// TwinCAT 3 PLC project Builder2
// ProgramVersion: 3.1.4023.0
// libraries:
//   Tc2_Standard, * (Beckhoff Automation GmbH)
//   Tc2_System, * (Beckhoff Automation GmbH)
//   Tc3_Module, * (Beckhoff Automation GmbH)
//   VisuSymbols,3.5.10.0,System
// project tree:
//   / Class Diagram_1.TcCD (not stored), ConcreteBuilder.TcPOU, Director.TcPOU, GlobalTextList.TcGTLO, ITF_Builder.TcIO, PlcTask.TcTTO, Product.TcPOU, Visualization Manager.TcVMO (not stored)
//   POUs/ MAIN.TcPOU
//   VISUs/ Visualization.TcVIS
// real-time tasks:
//   TASK PlcTask: cycle T#10ms, priority 20, ADS port 350

CONFIGURATION Builder2
    RESOURCE PLC ON TwinCAT3
        TASK PlcTask(INTERVAL := T#10ms, PRIORITY := 20);
        PROGRAM MAIN WITH PlcTask : MAIN;
    END_RESOURCE
END_CONFIGURATION

// ---- ITF_Builder.TcIO
///Builder interface to declare all needed parts to be built
INTERFACE ITF_Builder

///Illustrative method of the pattern to set the main part
METHOD Set_Main_Part
VAR_INPUT
	///Illustrative value (object because it is a TRING) to be set as a product part
	mainPart: STRING;
END_VAR
END_METHOD

///Illustrative method of the pattern to set the part1
METHOD Set_Part1
VAR_INPUT
	///Illustrative value (object because it is a TRING) to be set as a product part
	part1: STRING;
END_VAR
END_METHOD

///Illustrative method of the pattern to set the part2
METHOD Set_Part2
VAR_INPUT
	///Illustrative value (object because it is a TRING) to be set as a product part
	part2: STRING;
END_VAR
END_METHOD

///Illustrative method of the pattern to set the part3
METHOD Set_Part3
VAR_INPUT
	///Illustrative value (object because it is a TRING) to be set as a product part
	part3: STRING;
END_VAR
END_METHOD

END_INTERFACE

// ---- POUs/MAIN.TcPOU
PROGRAM MAIN
VAR
	///Arrays with the different specifications for the Client to choose
	arrayChassis: ARRAY[1..3] OF STRING := ['Red Chassis ', 'Black Chassis ', 'White Chassis '];
	arrayCarType: ARRAY[1..3] OF STRING := ['Sedan ', 'Hatchback ', 'Sport '];
	arrayMotor: ARRAY[1..3] OF STRING := ['Motor 1.4cc ', 'Motor 2.0cc ', 'Motor 2.5cc '];
	arrayTires: ARRAY[1..3] OF STRING := ['Aluminium tires ', 'Chrome plated tires ', 'Ligth aluminium tires '];
	///Temporary array to have a reference to the clients choice
	tempArray: ARRAY[1..4] OF STRING;
	///Boolean and integer values to receive data from the tables in the visualization element
	///The boolean value validates if the client has chosen a valid option
	bChassis: BOOL := FALSE;
	///The integer value hold the reference to the array of specifications
	iChassis: INT := 0;
	///Boolean and integer values to receive data from the tables in the visualization element
	///The boolean value validates if the client has chosen a valid option
	bCarType: BOOL := FALSE;
	///The integer value hold the reference to the array of specifications
	iCarType: INT := 0;
	///Boolean and integer values to receive data from the tables in the visualization element
	///The boolean value validates if the client has chosen a valid option
	bMotor: BOOL := FALSE;
	///The integer value hold the reference to the array of specifications
	iMotor: INT := 0;
	///Boolean and integer values to receive data from the tables in the visualization element
	///The boolean value validates if the client has chosen a valid option
	bTires: BOOL := FALSE;
	///The integer value hold the reference to the array of specifications
	iTires: INT := 0;
	///Boolean value to verify and respond to a client's request
	bRequest: BOOL := FALSE;
	///String variable to interact and respond to the client in the visualization element
	sMessageLog: STRING(500) := 'Waiting for your request';
	///A pointer to Poduct to dynamically create and delete product objects at the clients requests
	prod: POINTER TO Product;
	///A ConcreteBuilder instance to be passed to the Director and build the final Product objects
	aConcreteBuilder: ConcreteBuilder;
	///A Director instance that is instanciated with a ConcreteBuilder instance and the first specifications.
	/// later on in the program these specifications of the ConcreteBuilder instance will be changed dynamically
	{attribute 'old_input_assignments' := ''}
	aDirector: Director(concreteBuilder := aConcreteBuilder, specifications := tempArray);	
END_VAR

//The visualization element has 4 coloums in which the client must select an option from each coloum.
//Once the client has made its choice, He can then procede to validate its request.
//The bottom rectangle will handle all possible responses from the application to the client.

//If the client makes a request in the visualization element
IF bRequest
	THEN
	//We verify that the cliet has chosen all the required parts(All in this case)
	IF bChassis AND bCarType AND bMotor AND bTires
		THEN
		//If the client has sent a valir request, the builder notifies the client about the received request
		sMessageLog := 'Your red car is being built';
		//A new product object is created on demand
		prod := __NEW(Product);
		//The tempArray is modified to the special characteristics demanded from the client on the visualization element
		tempArray[1] := arrayChassis[iChassis];
		tempArray[2] := arrayCarType[iCarType];
		tempArray[3] := arrayMotor[iMotor];
		tempArray[4] := arrayTires[iTires];

		//The Director object receives the specifications for the new Product to be built
		aDirector(spected := tempArray);
		//The Product object request the construction to the Director.
		prod^ := aDirector.Construct();
		//The Builder's response after the Director object has handled the proper request
		sMessageLog := CONCAT( 'Your car has been built. It has: ', prod^.toString());
		//Once this reques has been handled, the request flag is set to FALSE
		bRequest := FALSE;
		//Once this reques has been handled, the Product object is deleted to free memory
		__DELETE(prod);
		
		//If the client did not choose all the required parts
		ELSE
			
		//The Builder responds
		sMessageLog := 'You need to select all the parts for your car';
		//Once this reques has been handled, the reques flag is set to FALSE
		bRequest := FALSE;
		
	END_IF

END_IF

END_PROGRAM

// ---- Product.TcPOU
///The class Product is just a plain blueprint of the components of the object to be built.
///The final Product may ot may not contain the all the Parts listed on the Product declaration
/// rather only the parts in the specifications sent by the client.
{attribute 'enable_dynamic_creation' := ''}
FUNCTION_BLOCK Product
VAR_INPUT
	///List of possible parts to be build in a final Product object
	mainPart: STRING;
	part1: STRING;
	part2: STRING;
	part3: STRING;
END_VAR

///Method to be used in the visualization element for an easier String handling
METHOD toString : STRING
VAR
	///Local variable to join together and store the pieces of String
	tempString: STRING;
END_VAR
//tempString joins together "Main Part" and "Part 1" of the Product object
tempString := CONCAT(THIS^.mainPart , THIS^.part1);
//tempString joins together its current value and "Part 2" of the Product object
tempString := CONCAT(tempString , THIS^.part2);
//tempString joins together its current value and "Part 3" of the Product object
tempString := CONCAT(tempString , THIS^.part3);
//The final result is sent as the output of this method
toString := tempString;
END_METHOD

END_FUNCTION_BLOCK

// ---- ConcreteBuilder.TcPOU
///This is the concrete builder class, reponsible for building the final product object
FUNCTION_BLOCK ConcreteBuilder IMPLEMENTS ITF_Builder
VAR
	///Holds an internal reference to how the final product shoud be so the builder class can build it on the fly 
	/// without any help from other classes exepting the Director class that is going to be passing the special
	///specifications to the builder.
	localProduct: Product;
END_VAR

///Illustrative method of the pattern to get the main part
METHOD Get_Main_Part : STRING
//Returns the object stored in the built product THIS^.localProduct.mainPart
Get_Main_Part := THIS^.localProduct.mainPart;
END_METHOD

///Illustrative method of the pattern to get the part1
METHOD Get_Part1 : STRING
//Returns the object stored in the built product THIS^.localProduct.part1
Get_Part1 := THIS^.localProduct.part1;
END_METHOD

///Illustrative method of the pattern to get the part2
METHOD Get_Part2 : STRING
//Returns the object stored in the built product THIS^.localProduct.part2
Get_Part2 := THIS^.localProduct.part2;
END_METHOD

///Illustrative method of the pattern to get the part3
METHOD Get_Part3 : STRING
//Returns the object stored in the built product THIS^.localProduct.part3
Get_Part3 := THIS^.localProduct.part3;
END_METHOD

///Illustrative method of the pattern
METHOD Get_Result : Product
//The concrete builder, after it builts the final object of class product, returns the 
// final product object 
Get_Result := THIS^.localProduct;
END_METHOD

///Illustrative method of the pattern to set the main part
METHOD Set_Main_Part
VAR_INPUT
	///Illustrative value (object because it is a TRING) to be set as a product part
	mainPart: STRING;
END_VAR
//Sets the passed value to its corresponding field. 
//We can say that the the final product is in process of being built.
//So this is a step into building the final product done by the builder.
THIS^.localProduct.mainPart := mainPart;
END_METHOD

///Illustrative method of the pattern to set the part1
METHOD Set_Part1
VAR_INPUT
	///Illustrative value (object because it is a TRING) to be set as a product part
	part1: STRING;
END_VAR
//Sets the passed value to its corresponding field. 
//We can say that the the final product is in process of being built.
//So this is a step into building the final product done by the builder.
THIS^.localProduct.part1 := part1;
END_METHOD

///Illustrative method of the pattern to set the part2
METHOD Set_Part2
VAR_INPUT
	///Illustrative value (object because it is a TRING) to be set as a product part
	part2: STRING;
END_VAR
//Sets the passed value to its corresponding field. 
//We can say that the the final product is in process of being built.
//So this is a step into building the final product done by the builder.
THIS^.localProduct.part2 := part2;
END_METHOD

///Illustrative method of the pattern to set the part3
METHOD Set_Part3
VAR_INPUT
	///Illustrative value (object because it is a TRING) to be set as a product part
	part3: STRING;
END_VAR
//Sets the passed value to its corresponding field. 
//We can say that the the final product is in process of being built.
//So this is a step into building the final product done by the builder.
THIS^.localProduct.part3 := part3;
END_METHOD

END_FUNCTION_BLOCK

// ---- Director.TcPOU
///The director class is responsible to delegate the construction of the final product object 
/// to a concrete builder object.
FUNCTION_BLOCK Director
VAR_INPUT
	///This variable is sent by the client as the specifications of the final product to be built.
	spected: ARRAY[1..4] OF STRING;
END_VAR
VAR
	///Holds a reference to the concrete builder object to send the specifications of the final product to it.
	concreteBuilder: ConcreteBuilder;
	///Stores the specifications, sent by the client, of the final product to be built.
	specifications: ARRAY[1..4] OF STRING;
END_VAR

//This dynamic constructor changes the previous specifications of the final product to be built
THIS^.specifications := THIS^.spected;

///This method is going to be called by the client when a new Product object must be built
METHOD Construct : Product
//The Director tells its concreteBuilder instance to build the final product step by step passing the specifications stored in the 
// array THIS^.specifications[1..4]

//Step 1 "Main Part"
THIS^.concreteBuilder.Set_Main_Part(THIS^.specifications[1]);
//Step 2 "Part 1"
THIS^.concreteBuilder.Set_Part1(THIS^.specifications[2]);
//Step 3 "Part 2"
THIS^.concreteBuilder.Set_Part2(THIS^.specifications[3]);
//Step 4 "Part 3"
THIS^.concreteBuilder.Set_Part3(THIS^.specifications[4]);

//Finally the concreteBuilder instance in the Director object delivers the final result as a Product object
Construct := THIS^.concreteBuilder.Get_Result();
END_METHOD

///This constructor is called at instanciation to store the inital specifications of the product to be built and 
/// the reference to the builder object.
METHOD fb_init
VAR_INPUT
	/// TRUE: the Retain-variables are initialized (reset warm / reset cold)
	bInitRetains: BOOL;
	/// TRUE  the instance will be copied to the copy-code afterward (online change)
	bInCopyCode: BOOL;
	///Reference to the builder that is going to be building the final product object.
	concreteBuilder: ConcreteBuilder;
	///Specifications, sent by the client, to be built on the final product object
	specifications: ARRAY[1..4] OF STRING;
END_VAR
//Stores the reference to which builder will be building the final product object in its own field THIS^.concreteBuilder
THIS^.concreteBuilder := concreteBuilder;

//Stores the specifications to build the final product object in its own field THIS^.specifications.
THIS^.specifications := specifications;
END_METHOD

END_FUNCTION_BLOCK

// ---- GlobalTextList.TcGTLO
TEXTLIST GlobalTextList
  801 = '%s'
  165 = 'Builder´s response'
  546 = 'Car type'
  100 = 'Car Type'
  545 = 'Chassis Colour'
  112 = 'Choose your customized Car'
  823 = 'choose Your new Car'
  278 = 'Make Request'
  547 = 'Motor dimensions'
  710 = 'Motor Dimensions'
  909 = 'The visualization element has 4 columns in which the client mus select an option from each column.\nOnce the client has made its choice, He can then procede to validate its request.\nThe bottom rectangle will handle all posible responses from the application to the client.'
  486 = 'The visualization element lets the client chose an option blueprint to build a Car\nOnce the client has chosen his prefered option, he can then procede to make the request of construction.\nThe bottom rectangle will handle all posible responses from the application to the client.'
  44 = 'Tires'
  548 = 'Wheels type'
END_TEXTLIST

// ---- VISUs/Visualization.TcVIS
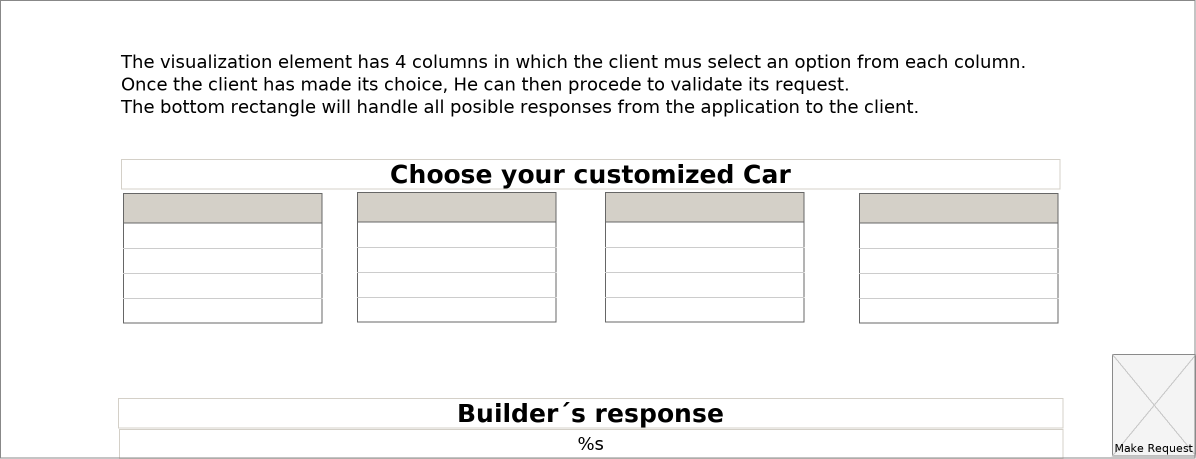
VISUALIZATION Visualization  // 1196x459
    Label (118,35 953x99), "The visualization element has 4 columns in which the client mus select an option from each column. Once the client has made its choice, He can then procede to validate its request. The bottom rectangle will handle all posible responses from the application to the client."
    Label (291,404 475x30)
    Image (1112,354 84x102), "Make Request", image: VisuSymbols.Symbols.OK
        OnMouseClick: toggle MAIN.bRequest
    Textfield (119,429 944x30), "%s", text variable: MAIN.sMessageLog
    Textfield (118,398 945x30), "Builder´s response"
    Textfield (121,159 939x30), "Choose your customized Car"
    Table (123,193 199x130), data array: MAIN.arrayChassis
        p3854506369: MAIN.arrayChassis[INDEX]
        p1892666644: MAIN.tableArray[2,INDEX]
        p338671338: MAIN.tableArray[3,INDEX]
        p2170511999: MAIN.tableArray[4,INDEX]
        p2232123230: Chassis Colour
        p511219082: Car type
        p1755163831: Motor dimensions
        p4092479075: Wheels type
        p1137915858: MAIN.iChassis
        p1822360349: MAIN.bChassis
    Table (357,192 199x130), data array: MAIN.arrayCarType
        p3854506369: MAIN.arrayCarType[INDEX]
        p1892666644: MAIN.tableArray[2,INDEX]
        p338671338: MAIN.tableArray[3,INDEX]
        p2170511999: MAIN.tableArray[4,INDEX]
        p2232123230: Car Type
        p511219082: Car type
        p1755163831: Motor dimensions
        p4092479075: Wheels type
        p1137915858: MAIN.iCarType
        p1822360349: MAIN.bCarType
    Table (605,192 199x130), data array: MAIN.arrayMotor
        p3854506369: MAIN.arrayMotor[INDEX]
        p1892666644: MAIN.tableArray[2,INDEX]
        p338671338: MAIN.tableArray[3,INDEX]
        p2170511999: MAIN.tableArray[4,INDEX]
        p2232123230: Motor Dimensions
        p511219082: Car type
        p1755163831: Motor dimensions
        p4092479075: Wheels type
        p1137915858: MAIN.iMotor
        p1822360349: MAIN.bMotor
    Table (859,193 199x130), data array: MAIN.arrayTires
        p3854506369: MAIN.arrayTires[INDEX]
        p1892666644: MAIN.tableArray[2,INDEX]
        p338671338: MAIN.tableArray[3,INDEX]
        p2170511999: MAIN.tableArray[4,INDEX]
        p511219082: Car type
        p1755163831: Motor dimensions
        p4092479075: Wheels type
        p1137915858: MAIN.iTires
        p1822360349: MAIN.bTires
END_VISUALIZATION
